FUNCTION_BLOCK Stage7 (* Template for a Basic Function Block Type *)
  (* Standard: 61499-2 *)
  (* Version 1.0, 2021-06-20, HP *)
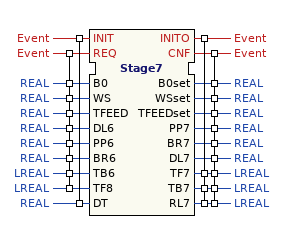
  EVENT_INPUT
    INIT WITH DT; (* Initialization Request *)
    REQ WITH B0, WS, TFEED, DL6, PP6, BR6, TB6, TF8; (* Normal Execution Request *)
  END_EVENT
  EVENT_OUTPUT
    INITO WITH TB7, RL7, TF7; (* Initialization Confirm *)
    CNF WITH TB7, DL7, TF7, BR7, PP7, TFEEDset, WSset, B0set, RL7; (* Execution Confirmation *)
  END_EVENT
  VAR_INPUT
    B0 : REAL;
    WS : REAL;
    TFEED : REAL;
    DL6 : REAL;
    PP6 : REAL;
    BR6 : REAL;
    TB6 : LREAL;
    TF8 : LREAL;
    DT : REAL;
  END_VAR
  VAR_OUTPUT
    B0set : REAL;
    WSset : REAL;
    TFEEDset : REAL;
    PP7 : REAL;
    BR7 : REAL;
    DL7 : REAL;
    TF7 : LREAL;
    TB7 : LREAL;
    RL7 : LREAL;
  END_VAR
  VAR
    AB : REAL; (* internal variabel *)
    UU : REAL;
    TREF : REAL;
    AD : REAL;
    AHC : REAL;
    AHR : REAL;
    AS : REAL;
    REC : REAL;
    WN : REAL;
    WN_1 : REAL;
    XKN : REAL;
    C1 : REAL;
    HS : REAL;
    G : REAL;
    W1 : REAL;
    TFREC : REAL;
    TS : REAL;
    DTS : REAL;
    TF7_last : REAL;
    RL7_last : REAL;
    TB7_last : REAL;
    USS : REAL;
    RHOB : REAL;
    CPB : REAL;
    CPF : REAL;
    FMW : REAL;
    HLV : REAL;
    HV : REAL;
    BPR : REAL;
    FMC : REAL;
    U : REAL;
    A : REAL;
    B : REAL;
    C : REAL;
    D1 : REAL;
    d : REAL;
    a : REAL;
    A1 : REAL;
    A2 : REAL;
    A3 : REAL;
    A4 : REAL;
    A5 : REAL;
    A6 : REAL;
    p : REAL;
    q : REAL;
    TC : REAL;
    PC : REAL;
    DTB7 : REAL;
    DEN7 : REAL;
    DH7 : REAL;
    DP7 : REAL;
    DPDH7 : REAL;
    DT7 : REAL;
    m : REAL;
    n : REAL;
    VR7 : REAL;
    DELTA7 : REAL;
    DELTA29 : REAL;
    DELTA51 : REAL;
    DELTA7_last : REAL;
    DELTA29_last : REAL;
    DELTA51_last : REAL;
  END_VAR
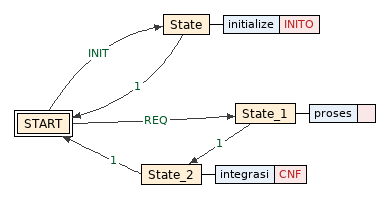
  EC_STATES
    START; (* Initial State *)
    State : initialize -> INITO;
    State_1 : proses;
    State_2 : integrasi -> CNF;
  END_STATES
  EC_TRANSITIONS
    START TO State := INIT;
    State TO START := 1;
    START TO State_1 := REQ;
    State_1 TO State_2 := 1;
    State_2 TO START := 1;
  END_TRANSITIONS
  ALGORITHM initialize IN ST: (* Initialization algorithm *)
TREF :=273.15;
AB :=57.2727;
AHC :=4069.2;
AHR :=2639.7;
AS :=3225.7;
REC :=0.0;
//TF2:=TF2;

//TFEED :=TFEED1+TREF;
 //TS:=TS1+TREF;
WN :=3.0;
XKN :=0.68;
HS:=0.11;
G :=9.81;
W1 :=0.50;

RL7 := 0.552127445016038;
TB7 := 348.429390583908;
TF7 := 344.515318586845;
TF8 := 341.885924485359;



RL7_last :=RL7;
TB7_last :=TB7;
TF7_last :=TF7;
  END_ALGORITHM
  ALGORITHM proses IN ST: (* kalkulasi *)
UU := TFEED;
U :=UU;

USS :=49.767;
C1 :=0.625;
RHOB :=1032.4; //maassa jenis brine
CPB :=1.00; //heatcapacity Brine
CPF :=1.00; //heat capacity feed
FMW :=23654.0;
HLV :=563.7959;
HV :=625.1971;
BPR :=2.192;
FMC :=34736.09;
//U :=UU; //feed temp



///  Calculate the physical properties

//A :=3.2437814;
//B :=5.86826*0.001;
//C :=1.1702379*0.00000001;
//D1 :=2.1878462*0.001;
//TC :=647.27;
//PC :=218.167;


A1 :=3.2437814;
A2:=5.86826*0.001;
A3:=1.1702379*0.00000001;
A4 :=2.1878462*0.001;
A5 :=647.27;
A6 :=218.167;

DTB7 :=A5-TB7;
DEN7 :=(A1+A2*DTB7+A3*DTB7*DTB7*DTB7)/(1+A4*DTB7)*DTB7/TB7;
p:=DEN7;
q:=10.0;
PP7 :=A6/(EXPT(q, p));

// calculate the brine flow rates
DP7:=PP6-PP7;
DH7:=RL7-C1*HS;
DPDH7 :=DP7*101000+G*RHOB*DH7;
m:=DPDH7*RHOB;
n:=0.5;
BR7 :=WN*XKN*RL7*(EXPT(m, n));
BR7 :=BR7*60.0/1000.0;

// calculate the vapor flow rates

DT7 :=TB7-BPR/1.8-(TF8+TF7)*0.5;
VR7 :=U*AHC*DT7/HLV/1000.0;
DL7 :=DL6+VR7;


//// state equation
DELTA7 :=(BR6-BR7-VR7)*1000.0/RHOB/AB;
DELTA29 :=((BR6*CPB*(TB6-TB7))-VR7*(HV-CPB*(TB7-TREF)))*1000.0/AB/RHOB/CPB/RL7;
DELTA51 :=(B0*CPF*(TF8-TF7)*1000+(U*AHC*DT7))/FMW/CPF;
  END_ALGORITHM
  ALGORITHM integrasi IN ST: (* new algorithm *)
B0set:=B0;
WSset:=WS ;
TFEEDset:=TFEED;
//integrasi
RL7 := (DELTA7 + DELTA7_last)*0.5*DT + RL7_last;
DELTA7_last :=DELTA7 ;
RL7_last :=RL7;

TB7:= (DELTA29 + DELTA29_last)*0.5*DT + TB7_last;
DELTA29_last :=DELTA29 ;
TB7_last:=TB7;

TF7 := (DELTA51 + DELTA51_last)*0.5*DT + TF7_last;
DELTA51_last :=DELTA51 ;
TF7_last :=TF7;
  END_ALGORITHM
END_FUNCTION_BLOCK
